FUNCTION_BLOCK PUBLIC FB_TimeControl
VAR_INPUT
	bEnable         :BOOL;
	bReset          :BOOL;
END_VAR
VAR_OUTPUT 
	nHour           :DINT;
	nMin            :DINT;
	nSec            :DINT;
	nTotalSec       :DINT;
END_VAR
VAR
	tpPulse1        :TP;
	tpPulse2        :TP;
	
	
    bMainStart      :BOOL;
    bStart1         :BOOL;
    bStart2         :BOOL;
    bStop           :BOOL;
    bPuls1          :BOOL;
    bPuls2          :BOOL;

    ftrigPuls1      :F_TRIG;
    ftrigPuls2      :F_TRIG;
    rtrigPulsMain   :R_TRIG;
	
	
END_VAR

rtrigPulsMain(CLK:= bEnable);
ftrigPuls1(CLK:= bPuls2);
ftrigPuls2(CLK:= bPuls1);

tpPulse1(IN:=(ftrigPuls1.Q OR rtrigPulsMain.Q) ,PT:= T#490MS);
bPuls1:= tpPulse1.Q;

tpPulse2(IN:=(ftrigPuls2.Q AND NOT bStop) ,PT:= T#490MS);
bPuls2:=tpPulse2.Q;

IF bEnable THEN
	bMainStart := TRUE;
ELSE 
	bMainStart := FALSE;
END_IF
bStop := NOT bMainStart;

IF bMainStart AND ftrigPuls1.Q THEN
	nTotalSec := nTotalSec + 1;
ELSIF bReset THEN
	nTotalSec := 0;
END_IF
//Secend
IF bMainStart AND ftrigPuls1.Q THEN
	nSec := nSec + 1;
	ELSIF (nSec = 60) THEN
	nSec := 0;
	ELSIF bReset THEN
	nSec := 0;	
END_IF
//Minutes
IF bMainStart THEN
	nMin := (nTotalSec-(nHour*3600)) /60;
	ELSIF bReset THEN
	nMin := 0;
END_IF
//Hours
IF bMainStart THEN
	nHour := nTotalSec/3600;
	ELSIF bReset THEN
	nHour := 0;
END_IF

END_FUNCTION_BLOCK

(* stored: Version 1.1.0.1, ProductVersion 3.1.4024.12
   POU FB_TimeControl: Id {61398d1a-2978-4106-99b0-e5770460c1f2}, SpecialFunc None *)
